# EPICS autosave request: dxpApp/Db/dxpSystem_settings.req
$(P)PollTime
$(P)NumSCAs
$(P)SaveSystemFile
$(P)MCARefreshPeriod
